FUNCTION_BLOCK Fb_SafetyCheck
VAR_INPUT
END_VAR
VAR_OUTPUT
END_VAR
VAR
	i, j:INT;
	m_checkDelay :ARRAY[1..g_maxNum] OF checkDelay;
	m_checkDelayTime :checkDelayTime;
	m_checkPermit:ARRAY[1..g_maxNum] OF  checkPermit;
	
	m_jntErrFlag:ARRAY[1..g_maxNum,0..g_maxArmJoint,1..3] OF BOOL;
	m_armErrFlag:ARRAY [1..g_maxNum,1..3] OF BOOL;
	m_errCode:UDINT;
	
	
	m_errNumType: ARRAY [1..3] OF INT;
	m_ArrayErrCodeType:ARRAY [1..3] OF ARRAY [0..30] OF UDINT;
	m_ArrayErrCodeTypeTest:ARRAY [1..3] OF ARRAY [0..100] OF UDINT;
	m_armErrCodePopup : ARRAY [1..4] OF ARRAY [0..2] OF UDINT;
	m_armErrCodeRefresh : ARRAY [1..4] OF UINT;
	
	//The fault is sent to the UI at the frequency of 0.1S
	m_errCodeUpdateFlag: ARRAY [1..3] OF BOOL;
	m_errCodeUpdateTon: ARRAY [1..3] OF TON;
	
	m_curJntTorqueIOlast :ARRAY [1..g_maxArmNum] OF vec13di;  
	m_cmdJntPosLast : ARRAY [1..g_maxArmNum] OF vec13d;  
	m_cartCurJntTorqueIOlast :vec8di;  
	m_cartCmdJntPosLast : vec8d;  
	o_ErrCode:ARRAY [1..3] OF UDINT;
		
	m_PromptMassBusy:BOOL;
	m_PromptFlag:ARRAY[1..g_maxNum,1..30] OF UINT;
	m_deleteCode:UDINT;
	
	//joint control error
	m_followErrLimit:vec13d:=[g_largeNum, g_largeNum, 0.010, 4(5*g_deg2Rad), 0.010, 5(170*g_deg2Rad)];
END_VAR


VAR CONSTANT
	m_codeUpdateDelay:TIME:=T#0.1S;
	
	//Fault level: 1 indicates  prompt message, 2 indicates a recoverable fault and 3 indicates an unrecoverable fault
	m_promptMessageLevel : UINT :=1;
	m_rcvLevel : UINT:=2;
	m_unrcvLevel : UINT :=3;
END_VAR

METHOD arrayDeleteFrist : ARRAY [0..30] OF UDINT;
VAR_INPUT
	i_array:ARRAY [0..30] OF UDINT;
END_VAR

VAR
	k:INT;
END_VAR

arrayDeleteFrist[30]:=0;

FOR k:=0 TO 29 BY 1 DO
	arrayDeleteFrist[k]:=i_array[k+1];
END_FOR
END_METHOD

METHOD arrayFILO : ARRAY [0..100] OF  UDINT
VAR_INPUT
	i_array:ARRAY[0..100] OF UDINT;
	i_newData:UDINT;
END_VAR

VAR
	i:INT;
END_VAR

FOR i:=0 TO 20 BY 1 DO
	arrayFILO[i]:=i_array[i];
	IF i_array[i]=0 THEN
		arrayFILO[i]:=i_newData;
		EXIT;
	END_IF
END_FOR
END_METHOD

METHOD cartSafetyCheck : BOOL
VAR_INPUT
	i_armId:UDINT;
	i_safetyCheckVar : checkInputVariable;
	i_cartJointData : ST_CartJointData;
END_VAR


VAR
	k:INT;
END_VAR


//驱动器状态监测、驱动器未连接
FOR i:=1 TO g_maxCartJoint BY 1 DO
	m_checkDelay[i_ArmId].T_cartJntStatusErr[i](IN:= (i_safetyCheckVar.m_cartDriverInput[i].m_statusWord=0 AND m_checkPermit[i_ArmId].m_cartJntStatus[i]), PT:=m_checkDelayTime.Ti_CarJntStatus , Q=> , ET=> );
	IF m_checkDelay[i_ArmId].T_cartJntStatusErr[i].Q THEN
		errCodeAssign(i_ArmId, i_ArmId+3,  0, i, 16#3002 ,m_unrcvLevel );
	END_IF
END_FOR



//关节编码器监测
FOR i:=1 TO g_maxCartJoint BY 1 DO
	m_checkDelay[i_ArmId].T_cartLinkEncErr[i](IN:= (i_safetyCheckVar.m_cartDriverInput[i].m_linkEncoder=g_cartMaxLinkEnc[i] OR i_safetyCheckVar.m_cartDriverInput[i].m_linkEncoder=g_cartMinLinkEnc[i]) AND m_checkPermit[i_ArmId].m_cartJntEncErr[i], PT:=m_checkDelayTime.Ti_CarActSec , Q=> , ET=> );
	IF m_checkDelay[i_ArmId].T_cartLinkEncErr[i].Q THEN
		errCodeAssign(i_ArmId, i_ArmId+3,  0, i, 16#3003 ,m_unrcvLevel );
	END_IF
END_FOR


//驱动器错误检测
FOR i:=1 TO g_maxCartJoint BY 1 DO
	m_checkDelay[i_ArmId].T_cartDriveErr[i](IN:= (i_safetyCheckVar.m_cartDriverInput[i].m_driverError AND 16#20)=32 AND m_checkPermit[i_ArmId].m_cartDriveErr[i] , PT:=m_checkDelayTime.Ti_CarDriveErr , Q=> , ET=> );
	IF m_checkDelay[i_ArmId].T_cartDriveErr[i].Q THEN
		errCodeAssign(i_ArmId, i_ArmId+3,  0, i, 16#3004 ,m_unrcvLevel );
	END_IF
END_FOR



//台车双编码器偏差过大
FOR i:=1 TO g_maxCartJoint BY 1 DO
	m_checkDelay[i_ArmId].T_cartJntEncErr[i](IN:= ABS (i_cartJointData.m_curLinkPos[i]-i_cartJointData.m_curJntPos[i])>g_cartMaxJntEncErr[i] AND m_checkPermit[i_ArmId].m_cartJntEncErr[i], PT:=m_checkDelayTime.Ti_CarDualEncDev , Q=> , ET=> );
	IF m_checkDelay[i_ArmId].T_cartJntEncErr[i].Q THEN
		errCodeAssign(i_ArmId, i_ArmId+3,  0, i, 16#3005 ,m_unrcvLevel );
	END_IF
END_FOR


//关节运动超限位
FOR i:=1 TO g_maxCartJoint BY 1 DO
	m_checkDelay[i_ArmId].T_cartOutOfLimit[i](IN:= (i_cartJointData.m_curJntPos[i]>=g_cartMaxJntPos[i] OR i_cartJointData.m_curJntPos[i]<=g_cartMinJntPos[i]) AND m_checkPermit[i_ArmId].m_cartOutOfLimit[i] , PT:=m_checkDelayTime.Ti_CaroutofLimit , Q=> , ET=> );
	IF m_checkDelay[i_ArmId].T_cartOutOfLimit[i].Q THEN
		errCodeAssign(i_ArmId, i_ArmId+3,  0, i, 16#3006 ,m_unrcvLevel );
	END_IF
END_FOR


//驱动器内部通讯错误
FOR i:=1 TO g_maxCartJoint BY 1 DO
	m_checkDelay[i_ArmId].T_cartCurrentIsNotUpdate[i](IN:= (i_safetyCheckVar.m_cartDriverInput[i].m_current=m_cartCurJntTorqueIOlast[i] AND m_checkPermit[i_ArmId].m_cartCurrentIsNotUpdate[i]), PT:=m_checkDelayTime.Ti_CarTorMotor , Q=> , ET=> );
	IF m_checkDelay[i_ArmId].T_cartCurrentIsNotUpdate[i].Q THEN
		errCodeAssign(i_ArmId, i_ArmId+3,  0, i, 16#3009 ,m_unrcvLevel );
	END_IF
	m_cartCurJntTorqueIOlast[i]:=i_safetyCheckVar.m_cartDriverInput[i].m_current;
END_FOR


//关节跟随误差过大
FOR i:=1 TO g_maxCartJoint BY 1 DO
	m_checkDelay[i_ArmId].T_cartJntFollowErr[i](IN:= ABS(i_cartJointData.m_cmdJntPos[i]- i_cartJointData.m_curJntPos[i])>g_cartMaxJntFollowErr[i]  AND m_checkPermit[i_ArmId].m_cartFollowErr[i], PT:=m_checkDelayTime.Ti_CarFollowDev , Q=> , ET=> );
	IF m_checkDelay[i_ArmId].T_cartJntFollowErr[i].Q THEN
		errCodeAssign(i_ArmId, i_ArmId+3,  0, i, 16#2002 ,m_rcvLevel );
	END_IF
END_FOR


//关节速度监控
FOR i:=1 TO g_maxCartJoint BY 1 DO
	m_checkDelay[i_ArmId].T_cartJntVelErr[i](IN:= ABS(i_cartJointData.m_curJntVel[i])>g_cartMaxJntVel[i] AND m_checkPermit[i_ArmId].m_cartJntVelErr[i], PT:=m_checkDelayTime.Ti_CarJntVel , Q=> , ET=> );
	IF m_checkDelay[i_ArmId].T_cartJntVelErr[i].Q THEN
		errCodeAssign(i_ArmId, i_ArmId+3,  0, i, 16#2003 ,m_rcvLevel );
	END_IF
END_FOR


//电流超限监测
FOR i:=1 TO g_maxCartJoint BY 1 DO
	m_checkDelay[i_ArmId].T_cartJntCurrentErr[i](IN:= ABS(i_cartJointData.m_curJntTrq[i])>g_cartMaxJntCurrent[i] AND m_checkPermit[i_ArmId].m_cartJntCurrentErr[i], PT:=m_checkDelayTime.Ti_CarJntCurrent , Q=> , ET=> );
	IF m_checkDelay[i_ArmId].T_cartJntCurrentErr[i].Q THEN
		errCodeAssign(i_ArmId, i_ArmId+3,  0, i, 16#2005 ,m_rcvLevel );
	END_IF
END_FOR


//Ethercat通讯检测
FOR i:=1 TO g_maxCartJoint BY 1 DO
	IF NOT i_safetyCheckVar.m_cartEtherCATState[i].EtherCATState THEN
		errCodeAssign(i_ArmId, i_ArmId+3,  0, i, 16#2006 ,m_rcvLevel );
	END_IF
END_FOR


//鸣志驱动器错误检测
FOR i:=1 TO g_maxCartJoint BY 1 DO
	m_checkDelay[i_ArmId].T_CarMingzhiDriveErr[i](IN:= (i_safetyCheckVar.m_cartDriverInput[i].m_statusWord AND 16#0F)=15  AND m_checkPermit[i_ArmId].m_cartMZDriveErr[i] , PT:=m_checkDelayTime.Ti_CarMZDriveErr , Q=> , ET=> );
	IF m_checkDelay[i_ArmId].T_CarMingzhiDriveErr[i].Q THEN
		errCodeAssign(i_ArmId, i_ArmId+3,  0, i, 16#2009 ,m_rcvLevel );
	END_IF
END_FOR
END_METHOD

PROPERTY checkPermit : REFERENCE TO ARRAY[1..g_maxNum] OF  checkPermit
GET
checkPermit ref= m_checkPermit;
END_GET
SET
END_SET
END_PROPERTY

METHOD electriAngleDev : DINT
VAR_INPUT
	i_motorElectriAngleDev : DINT;
END_VAR

IF i_motorElectriAngleDev > 50000 THEN
	electriAngleDev := i_motorElectriAngleDev - 65535;
ELSIF i_motorElectriAngleDev < -50000 THEN
	electriAngleDev := i_motorElectriAngleDev + 65535;
ELSE
	electriAngleDev := i_motorElectriAngleDev;
END_IF
END_METHOD

METHOD errCodeAssign : BOOL
VAR_INPUT
	i_armId:UDINT;
	i_errLocation:UDINT;
	i_errCodeMode:UDINT;
	i_errJoint:UDINT;
	i_errID:UDINT;
	i_errFlagID :UINT;
END_VAR
IF m_jntErrFlag[i_armId,i_errJoint,i_errFlagID]=FALSE THEN
	m_jntErrFlag[i_armId,i_errJoint,i_errFlagID]:=TRUE;
	m_errCode:=SHL(i_errLocation,24)+SHL(i_errCodeMode,20)+SHL(i_errJoint,16)+i_errID;
	
	
	IF i_errID>=16#3000 THEN
		m_errNumType[m_unrcvLevel]:=LIMIT(0,m_errNumType[m_unrcvLevel]+1,100);
		m_arrayErrCodeType[m_unrcvLevel][m_errNumType[m_unrcvLevel]]:=m_errCode;
		g_arrayErrCodeArm[i_armId]:=arrayFILO(i_Array:= g_arrayErrCodeArm[i_ArmId], i_NewData:=m_errCode );
		m_armErrFlag[i_armId,m_unrcvLevel]:=TRUE;
		
	ELSIF i_errID>=16#2000 THEN
		m_errNumType[m_rcvLevel]:=LIMIT(0,m_errNumType[m_rcvLevel]+1,100);
		m_arrayErrCodeType[m_rcvLevel][m_errNumType[m_rcvLevel]]:=m_errCode;
		g_arrayErrCodeArm[i_armId]:=arrayFILO(i_Array:= g_arrayErrCodeArm[i_ArmId], i_NewData:=m_errCode );
		m_armErrFlag[i_armId,m_rcvLevel]:=TRUE;
		
	END_IF
END_IF
END_METHOD

METHOD errCodeUpdating :ARRAY [1..3] OF UDINT;
VAR_INPUT
END_VAR

m_errCodeUpdateTon[m_unrcvLevel](IN:= NOT m_errCodeUpdateFlag[3], PT:=m_codeUpdateDelay , Q=> m_errCodeUpdateFlag[3], ET=> );
IF m_errCodeUpdateFlag[m_unrcvLevel] THEN
	IF m_errNumType[m_unrcvLevel]>=1 THEN
		m_ArrayErrCodeType[m_unrcvLevel]:=ArrayDeleteFrist(i_Array:=m_ArrayErrCodeType[3]) ;
		o_ErrCode[m_unrcvLevel]:=m_ArrayErrCodeType[m_unrcvLevel][0] ;
		m_ArrayErrCodeTypeTest[m_unrcvLevel]:=arrayFILO(i_Array:= m_ArrayErrCodeTypeTest[m_unrcvLevel], i_NewData:=o_ErrCode[m_unrcvLevel] );
		m_errNumType[m_unrcvLevel]:=m_errNumType[m_unrcvLevel]-1;
	END_IF
END_IF


m_errCodeUpdateTon[m_rcvLevel](IN:= NOT m_errCodeUpdateFlag[m_rcvLevel], PT:=m_codeUpdateDelay , Q=> m_errCodeUpdateFlag[2], ET=> );
IF m_errCodeUpdateFlag[m_rcvLevel] THEN
	IF m_errNumType[m_rcvLevel]>=1 THEN
		m_ArrayErrCodeType[m_rcvLevel]:=ArrayDeleteFrist(i_Array:=m_ArrayErrCodeType[2]) ;
		o_ErrCode[m_rcvLevel]:=m_ArrayErrCodeType[m_rcvLevel][0] ;
		m_ArrayErrCodeTypeTest[m_rcvLevel]:=arrayFILO(i_Array:= m_ArrayErrCodeTypeTest[m_rcvLevel], i_NewData:=o_ErrCode[m_rcvLevel] );
		m_errNumType[m_rcvLevel]:=m_errNumType[m_rcvLevel]-1;
	END_IF
END_IF
END_METHOD

METHOD errFlagReset : BOOL
VAR_INPUT
END_VAR

FOR i := 1 TO g_maxNum DO
	FOR j :=0 TO g_maxArmJoint DO
		m_jntErrFlag[i, j, 2]:=FALSE;
	END_FOR
	m_armErrFlag[i, 2]:=FALSE;
END_FOR

o_ErrCode[2]:=0;
END_METHOD

METHOD poseErrCheck : vec6d
VAR_INPUT
	i_cmdPose : ST_Frame;
	i_curPose :ST_Frame;
END_VAR

VAR
	posErr,oriErr:Vec3d;
	matT,rotErr:Mat3d;
	errAngle :LREAL;
	errAxis :Vec3d;
	i : INT;
END_VAR
vecSub(i_cmdPose.m_pos, i_curPose.m_pos,posErr);

matTranspose(i_cmdPose.m_rot, matT);
matMultiply(matT,i_curPose.m_rot, rotErr);
rot2AngAxis(rotErr, angle=>errAngle, axis=>errAxis);
vecMultiNum(errAxis, errAngle,oriErr);

FOR i := 1 TO 6 DO
	IF i <= 3 THEN
		poseErrCheck[i] := posErr[i];
	ELSE
		poseErrCheck[i] := oriErr[i];
	END_IF
END_FOR
END_METHOD

METHOD promptMassCode : BOOL
VAR_INPUT
	i_PromptStatus:BOOL;
	i_ArmId:UDINT;
	i_ErrID:UDINT;
	i_ErrLocation:UDINT;
END_VAR
VAR
	m_errStatus : UDINT := 0;
	//error ID , 0-15 bit
	m_errId : UDINT;
	m_arrayErrCode : ARRAY [0..30] OF UDINT;
	m_armErrCode : ARRAY [0..2] OF UDINT;
END_VAR

m_PromptMassBusy:=TRUE;

//prompt flag set true
IF i_PromptStatus=TRUE AND m_PromptFlag[i_ArmId,i_ErrID]=0 THEN
	m_PromptFlag[i_ArmId,i_ErrID]:=1;
END_IF

//
IF i_ErrLocation <= 7 AND i_ErrLocation >= 4 THEN
	m_errStatus := 16#00FF;
ELSE
	m_errStatus := 0;
END_IF
m_errId := i_errID+16#1020;

//output prompt error code
IF m_PromptFlag[i_ArmId,i_ErrID]=1 THEN
	m_ErrCode:=SHL(i_ErrLocation,24)+SHL(m_errStatus,16)+i_errID+16#1020;
	vecFIFO(m_ArrayErrCodeType[1] , m_ErrCode , m_arrayErrCode );
	m_ArrayErrCodeType[1]:=m_arrayErrCode;
	IF (m_ErrCode AND 16#00FF0000) = 16#00FF0000 THEN
		vecFIFO(m_armErrCodePopup[i_armId] , m_ErrCode , m_armErrCode );
		m_armErrCodePopup[i_armId] := m_armErrCode;
		m_armErrCodeRefresh[i_armId] := 1;
	END_IF
	m_PromptFlag[i_ArmId,i_ErrID]:=2;
END_IF

//clear prompt error code
IF m_PromptFlag[i_ArmId,i_ErrID]=2 AND i_PromptStatus=FALSE THEN
	m_deleteCode:=SHL(i_ErrLocation,24)+SHL(m_errStatus,16)+i_ErrID+16#1020;
	vecDeleteInput(m_ArrayErrCodeType[1] , m_deleteCode , m_arrayErrCode);
	m_ArrayErrCodeType[1] := m_arrayErrCode;
	IF (m_deleteCode AND 16#00FF0000)  = 16#00FF0000 THEN
		vecDeleteInput(m_armErrCodePopup[i_armId] , m_deleteCode , m_armErrCode );
		m_armErrCodePopup[i_armId] := m_armErrCode;
		m_armErrCodeRefresh[i_armId] := 2;
	END_IF
	//ArrayDeleteInput(i_Array:= m_ArrayErrCodeType[1], i_DeleteCode:=m_deleteCode , o_Array=> m_ArrayErrCodeType[1]);
	m_PromptFlag[i_ArmId,i_ErrID]:=0;
END_IF
o_ErrCode[1]:=m_ArrayErrCodeType[1][0];
m_PromptMassBusy:=FALSE;
END_METHOD

METHOD rcpErrCheck : BOOL
VAR_INPUT
	i_cmdPos : Vec3d;
	i_curPos : Vec3d;
END_VAR
VAR_IN_OUT
	r_errCount:INT;
	r_posErr :Vec3d;
END_VAR

VAR
	err:Vec3d;
END_VAR
vecSub(i_cmdPos, i_curPos,err);
r_posErr:=err;

IF  (norm(err)>g_rcpDeviationThres) THEN
	r_errCount:= r_errCount +1;
ELSE 
	r_errCount:=0;
END_IF
rcpErrCheck := r_errCount >= g_faultTriggerCounts;
END_METHOD

METHOD setupSafetyCheck : BOOL
VAR_INPUT
	i_armId:UDINT;
	i_safetyCheckVar :ARRAY[1..g_maxNum] OF checkInputVariable;
	i_setupJointData : ST_SetupJointData;
END_VAR

VAR
	k:INT;
END_VAR


//驱动器状态监测、驱动器未连接
FOR i:=1 TO g_setupJntNum BY 1 DO
	m_checkDelay[i_ArmId].T_jntStatusErr[i](IN:= (i_safetyCheckVar[i_ArmId].m_setupDriverInput[i].m_statusWord=0 AND m_checkPermit[i_ArmId].m_jntStatusErr[i]), PT:=m_checkDelayTime.Ti_jntStatusErr , Q=> , ET=> );
	IF m_checkDelay[i_ArmId].T_jntStatusErr[i].Q THEN
		errCodeAssign(i_ArmId, i_ArmId+3,  0, i, 16#3002 ,m_unrcvLevel );
	END_IF
END_FOR



//关节编码器监测
FOR i:=1 TO g_setupJntNum BY 1 DO
	m_checkDelay[i_ArmId].T_linkEncErr[i](IN:= (i_safetyCheckVar[i_ArmId].m_setupDriverInput[i].m_linkEncoder=g_maxLinkEnc[i] OR i_safetyCheckVar[i_ArmId].m_setupDriverInput[i].m_linkEncoder=g_minLinkEnc[i]) AND m_checkPermit[i_ArmId].m_linkEncErr[i], PT:=m_checkDelayTime.Ti_linkEncErr , Q=> , ET=> );
	IF m_checkDelay[i_ArmId].T_linkEncErr[i].Q THEN
		errCodeAssign(i_ArmId, i_ArmId+3,  0, i,  16#3003 ,m_unrcvLevel );
	END_IF
END_FOR


//驱动器错误检测
FOR i:=1 TO g_setupJntNum BY 1 DO
	m_checkDelay[i_ArmId].T_DriveErr[i](IN:= (i_safetyCheckVar[i_ArmId].m_setupDriverInput[i].m_driverError AND 16#20)=g_driveErrWord AND m_checkPermit[i_ArmId].m_driveErr[i] , PT:=m_checkDelayTime.Ti_driveErr , Q=> , ET=> );
	IF m_checkDelay[i_ArmId].T_DriveErr[i].Q THEN
		errCodeAssign(i_ArmId, i_ArmId+3,  0, i, 16#3004 ,m_unrcvLevel );
	END_IF
END_FOR


//双编码器偏差过大检测
FOR i:=1 TO g_setupJntNum BY 1 DO
	m_checkDelay[i_ArmId].T_armJntEncErr[i](IN:= ABS(i_setupJointData.m_curLinkPos[i_armId][i]-i_setupJointData.m_curJntPos[i_armId][i])>=g_armMaxJntEncErr[i] AND m_checkPermit[i_ArmId].m_armJntEncErr[i], PT:=m_checkDelayTime.Ti_armJntEncErr , Q=> , ET=> );
	IF m_checkDelay[i_ArmId].T_armJntEncErr[i].Q THEN
		errCodeAssign( i_ArmId, i_ArmId+3,  0, i, 16#3005, m_unrcvLevel );
	END_IF
END_FOR


//关节运动超限位
FOR i:=1 TO g_setupJntNum BY 1 DO
	m_checkDelay[i_ArmId].T_outOfLimit[i](IN:= (i_setupJointData.m_curJntPos[i_armId][i]>=(g_maxJntPos[i_armId,i]+g_armJntPosLimitBuffer[i]) OR i_setupJointData.m_curJntPos[i_armId][i]<=(g_minJntPos[i_armId,i]-g_armJntPosLimitBuffer[i])) AND m_checkPermit[i_ArmId].m_outOfLimit[i] , PT:=m_checkDelayTime.Ti_outofLimit , Q=> , ET=> );
	IF m_checkDelay[i_ArmId].T_outOfLimit[i].Q THEN
		errCodeAssign(i_ArmId, i_ArmId+3,  0, i, 16#3006, m_unrcvLevel );
	END_IF
END_FOR


//电机电角度偏差
FOR i:=1 TO g_setupJntNum BY 1 DO
	IF ABS(electriAngleDev(i_safetyCheckVar[i_armId].m_setupDriverInput[i].m_electriAngleDev))> g_motPhieErrLimit  AND m_checkPermit[i_ArmId].m_motPhieErr[i] THEN
		errCodeAssign(i_ArmId, i_ArmId+3,  0, i, 16#3008, m_unrcvLevel );
	END_IF
END_FOR


//驱动器内部通讯错误
FOR i:=1 TO g_setupJntNum BY 1 DO
	m_checkDelay[i_ArmId].T_currentIsNotUpdate[i](IN:= (i_safetyCheckVar[i_ArmId].m_setupDriverInput[i].m_current=m_curJntTorqueIOlast[i_ArmId][i] AND m_checkPermit[i_ArmId].m_currentIsNotUpdate[i]), PT:=m_checkDelayTime.Ti_currentIsNotUpdate , Q=> , ET=> );
	IF  m_checkDelay[i_ArmId].T_currentIsNotUpdate[i].Q THEN
		errCodeAssign(i_ArmId, i_ArmId+3,  0, i, 16#3009 ,m_unrcvLevel );
	END_IF
	m_curJntTorqueIOlast[i_ArmId][i]:=i_safetyCheckVar[i_ArmId].m_setupDriverInput[i].m_current;
END_FOR


//关节跟随误差过大
FOR i:=1 TO g_setupJntNum BY 1 DO
	m_checkDelay[i_ArmId].T_armJntFollowErr[i](IN:= ABS(i_setupJointData.m_cmdJntPos[i_armId][i]- i_setupJointData.m_curJntPos[i_armId][i])>g_armMaxJntFollowErr[i]  AND m_checkPermit[i_ArmId].m_armJntFollowErr[i], PT:=m_checkDelayTime.Ti_armJntFollowErr , Q=> , ET=> );
	IF m_checkDelay[i_ArmId].T_armJntFollowErr[i].Q THEN
		errCodeAssign(i_ArmId, i_ArmId+3,  0, i, 16#2002, m_rcvLevel );
	END_IF
END_FOR


//关节速度监控
FOR i:=1 TO g_setupJntNum BY 1 DO
	m_checkDelay[i_ArmId].T_jntVelErr[i](IN:= ABS (i_setupJointData.m_curJntVel[i_armId][i])>g_safetyJntVel[i] AND m_checkPermit[i_ArmId].m_jntVelErr[i], PT:=m_checkDelayTime.Ti_jntVelErr , Q=> , ET=> );
	IF m_checkDelay[i_ArmId].T_jntVelErr[i].Q THEN
		errCodeAssign(i_ArmId, i_ArmId+3,  0, i, 16#2003, m_rcvLevel );
	END_IF
END_FOR



//电流超限监测
FOR i:=1 TO g_setupJntNum BY 1 DO
	m_checkDelay[i_ArmId].T_jntCurrentErr[i](IN:= ABS(i_setupJointData.m_rawJntCurrent[i_armId][i])>g_maxJntCurrent[i] AND m_checkPermit[i_ArmId].m_jntCurrentErr[i], PT:=m_checkDelayTime.Ti_jntCurrentErr , Q=> , ET=> );
	IF m_checkDelay[i_ArmId].T_jntCurrentErr[i].Q THEN
		errCodeAssign(i_ArmId, i_ArmId+3,  0, i, 16#2005, m_rcvLevel );
	END_IF
END_FOR


//Ethercat通讯检测
FOR i:=1 TO g_setupJntNum BY 1 DO
	IF NOT i_safetyCheckVar[i_ArmId].m_EtherCATState[i].EtherCATState THEN
		errCodeAssign(i_ArmId, i_ArmId+3, 0, i, 16#2006, m_rcvLevel );
	END_IF
END_FOR


//不动点发生变化监控
m_checkDelay[i_ArmId].T_FixedPointErr(IN:=  i_safetyCheckVar[i_ArmId].m_rcpCheck AND m_checkPermit[i_ArmId].m_fixedPointErr, PT:=m_checkDelayTime.Ti_FixedPointErr , Q=> , ET=> );
IF m_checkDelay[i_ArmId].T_FixedPointErr.Q THEN
	errCodeAssign(i_ArmId, i_ArmId+3,  0, 0, 16#2007, m_rcvLevel );
END_IF


//目标位置指令突变检测
FOR i:=1 TO g_setupJntNum BY 1 DO
	IF (i_setupJointData.m_cmdJntPos[i_armId][i]-m_cmdJntPosLast[i_ArmId][i])>g_maxJntCmdSalta[i] AND m_checkPermit[i_ArmId].m_cmdJntSaltation[i] THEN
		errCodeAssign(i_armId, i_ArmId+3, 0, i, 16#2008, m_rcvLevel );
	END_IF
	m_cmdJntPosLast[i_armId][i] := i_setupJointData.m_cmdJntPos[i_armId][i];
END_FOR


//Deviation between command current and feedback current
FOR i:=1 TO g_setupJntNum BY 1 DO
	IF ABS(i_safetyCheckVar[i_armId].m_slaveDriverOutput[i].m_cmdCurrent-i_safetyCheckVar[i_armId].m_slaveDriverInput[i].m_current)> g_jntCurrentCtrlLimit[i]  AND m_checkPermit[i_armId].m_jntCurrentCtrlErr[i] THEN
		errCodeAssign(i_armId, i_armId+3, 0, i, 16#200B, m_rcvLevel );
	END_IF
END_FOR


//motor encoder mutation detection
FOR i:=1 TO g_setupJntNum BY 1 DO
	IF (i_safetyCheckVar[i_armId].m_motorEncoderSaltaValue[i])>g_maxJntCurSalta[i] THEN
		errCodeAssign(i_armId, i_ArmId+3, 0, i, 16#200C, m_rcvLevel );
	END_IF
END_FOR
END_METHOD

METHOD slaveSafetyCheck : BOOL
VAR_INPUT
	i_armId:UDINT;
	i_safetyCheckVar :ARRAY[1..g_maxNum] OF checkInputVariable;
	i_slaveJointData : ST_SlaveJointData;
END_VAR
//驱动器状态监测、驱动器未连接
FOR i:=1 TO g_sJntNum BY 1 DO
	m_checkDelay[i_ArmId].T_jntStatusErr[i+g_setupJntNum](IN:= (i_safetyCheckVar[i_ArmId].m_slaveDriverInput[i].m_statusWord=0 AND m_checkPermit[i_ArmId].m_jntStatusErr[i+g_setupJntNum]), PT:=m_checkDelayTime.Ti_jntStatusErr , Q=> , ET=> );
	IF m_checkDelay[i_ArmId].T_jntStatusErr[i+g_setupJntNum].Q  THEN
		errCodeAssign(i_ArmId, i_ArmId+3,  0, i+g_setupJntNum, 16#3002 ,m_unrcvLevel );
	END_IF
END_FOR



//关节编码器监测
FOR i:=1 TO g_sJntNum BY 1 DO
	m_checkDelay[i_ArmId].T_linkEncErr[i+g_setupJntNum](IN:= (i_safetyCheckVar[i_ArmId].m_slaveDriverInput[i].m_linkEncoder=g_maxLinkEnc[i] OR i_safetyCheckVar[i_ArmId].m_slaveDriverInput[i].m_linkEncoder=g_minLinkEnc[i]) AND m_checkPermit[i_ArmId].m_linkEncErr[i], PT:=m_checkDelayTime.Ti_linkEncErr , Q=> , ET=> );
	IF m_checkDelay[i_ArmId].T_linkEncErr[i+g_setupJntNum].Q THEN
		errCodeAssign(i_ArmId, i_ArmId+3,  0, i+g_setupJntNum,  16#3003 ,m_unrcvLevel );
	END_IF
END_FOR


//驱动器错误检测
FOR i:=1 TO g_sJntNum BY 1 DO
	m_checkDelay[i_ArmId].T_DriveErr[i+g_setupJntNum](IN:= (i_safetyCheckVar[i_ArmId].m_slaveDriverInput[i].m_driverError AND 16#20)=g_driveErrWord AND m_checkPermit[i_ArmId].m_driveErr[i] , PT:=m_checkDelayTime.Ti_driveErr , Q=> , ET=> );
	IF m_checkDelay[i_ArmId].T_DriveErr[i+g_setupJntNum].Q THEN
		errCodeAssign(i_ArmId, i_ArmId+3,  0, i+g_setupJntNum, 16#3004 ,m_unrcvLevel );
	END_IF
END_FOR


//双编码器偏差过大检测
FOR i:=1 TO g_sJntNum-5 BY 1 DO
	m_checkDelay[i_ArmId].T_armJntEncErr[i+g_setupJntNum](IN:= ABS(i_slaveJointData.m_curLinkPos[i_armId][i]-i_slaveJointData.m_curJntPos[i_armId][i])>=g_armMaxJntEncErr[i+g_setupJntNum] AND m_checkPermit[i_ArmId].m_armJntEncErr[i+g_setupJntNum], PT:=m_checkDelayTime.Ti_armJntEncErr , Q=> , ET=> );
	IF m_checkDelay[i_ArmId].T_armJntEncErr[i+g_setupJntNum].Q THEN
		errCodeAssign( i_ArmId, i_ArmId+3,  0, i+g_setupJntNum, 16#3005, m_unrcvLevel );
	END_IF
END_FOR


//关节运动超限位
FOR i:=1 TO g_sJntNum BY 1 DO
	m_checkDelay[i_ArmId].T_outOfLimit[i+g_setupJntNum](IN:= (i_slaveJointData.m_curJntPos[i_armId][i]>=(g_maxJntPos[i_armId,i+g_setupJntNum]+g_armJntPosLimitBuffer[i+g_setupJntNum]) OR i_slaveJointData.m_curJntPos[i_armId][i]<=(g_minJntPos[i_armId,i+g_setupJntNum]-g_armJntPosLimitBuffer[i+g_setupJntNum])) AND m_checkPermit[i_ArmId].m_outOfLimit[i+g_setupJntNum] , PT:=m_checkDelayTime.Ti_outofLimit , Q=> , ET=> );
	IF m_checkDelay[i_ArmId].T_outOfLimit[i+g_setupJntNum].Q THEN
		errCodeAssign(i_ArmId, i_ArmId+3,  0, i+g_setupJntNum, 16#3006, m_unrcvLevel );
	END_IF
END_FOR


//电机电角度偏差
FOR i:=1 TO g_sJntNum BY 1 DO
	IF ABS(electriAngleDev(i_safetyCheckVar[i_armId].m_slaveDriverInput[i].m_electriAngleDev))> g_motPhieErrLimit  AND m_checkPermit[i_ArmId].m_motPhieErr[i+g_setupJntNum] THEN
		errCodeAssign(i_ArmId, i_ArmId+3,  0, i+g_setupJntNum, 16#3008, m_unrcvLevel );
	END_IF
END_FOR


//驱动器内部通讯错误
FOR i:=1 TO g_sJntNum BY 1 DO
	m_checkDelay[i_ArmId].T_currentIsNotUpdate[i+g_setupJntNum](IN:= (i_safetyCheckVar[i_ArmId].m_slaveDriverInput[i].m_current=m_curJntTorqueIOlast[i_ArmId][i+g_setupJntNum] AND m_checkPermit[i_ArmId].m_currentIsNotUpdate[i+g_setupJntNum]), PT:=m_checkDelayTime.Ti_currentIsNotUpdate , Q=> , ET=> );
	IF  m_checkDelay[i_ArmId].T_currentIsNotUpdate[i+g_setupJntNum].Q THEN
		errCodeAssign(i_ArmId, i_ArmId+3,  0, i+g_setupJntNum, 16#3009 ,m_unrcvLevel );
	END_IF
	m_curJntTorqueIOlast[i_ArmId][i+g_setupJntNum]:=i_safetyCheckVar[i_ArmId].m_slaveDriverInput[i].m_current;
END_FOR


//关节跟随误差过大---1028
FOR i:=1 TO g_sJntNum BY 1 DO
	(*
	m_checkDelay[i_ArmId].T_armJntFollowErr[i+g_setupJntNum](IN:= ABS(i_slaveJointData.m_cmdJntPos[i_armId][i]- i_slaveJointData.m_curJntPos[i_armId][i])>g_armMaxJntFollowErr[i+g_setupJntNum]  AND m_checkPermit[i_ArmId].m_armJntFollowErr[i+g_setupJntNum], PT:=m_checkDelayTime.Ti_armJntFollowErr , Q=> , ET=> );
	IF m_checkDelay[i_ArmId].T_armJntFollowErr[i+g_setupJntNum].Q THEN
		errCodeAssign(i_ArmId, i_ArmId+3,  0, i+g_setupJntNum, 16#2002, m_rcvLevel );
	END_IF
	*)
	
	//update the control error limit
	IF (SlaveArmControl.m_slaveRobot.m_stiffChanged[i_ArmId]=TRUE) THEN
		m_followErrLimit:=g_armMaxJntFollowErrSoftStiff;
	ELSE
		m_followErrLimit:=g_armMaxJntFollowErr;
	END_IF
	
	//check
	m_checkDelay[i_ArmId].T_armJntFollowErr[i+g_setupJntNum](IN:= ABS(i_slaveJointData.m_cmdJntPos[i_armId][i]- i_slaveJointData.m_curJntPos[i_armId][i])>m_followErrLimit[i+g_setupJntNum]  AND m_checkPermit[i_ArmId].m_armJntFollowErr[i+g_setupJntNum], PT:=m_checkDelayTime.Ti_armJntFollowErr , Q=> , ET=> );
	IF m_checkDelay[i_ArmId].T_armJntFollowErr[i+g_setupJntNum].Q THEN
		errCodeAssign(i_ArmId, i_ArmId+3,  0, i+g_setupJntNum, 16#2002, m_rcvLevel );
	END_IF	
END_FOR


//关节速度监控
FOR i:=1 TO g_sJntNum-5 BY 1 DO
	m_checkDelay[i_ArmId].T_jntVelErr[i+g_setupJntNum](IN:= ABS (i_slaveJointData.m_curJntVel[i_armId][i])>g_safetyJntVel[i+g_setupJntNum] AND m_checkPermit[i_ArmId].m_jntVelErr[i+g_setupJntNum], PT:=m_checkDelayTime.Ti_jntVelErr , Q=> , ET=> );
	IF m_checkDelay[i_ArmId].T_jntVelErr[i+g_setupJntNum].Q THEN
		errCodeAssign(i_ArmId, i_ArmId+3,  0, i+g_setupJntNum, 16#2003, m_rcvLevel );
	END_IF
END_FOR


// TODO: replaced with cartesin twist check
//笛卡尔空间指令与位置偏差检测
//FOR i:=1 TO 6 BY 1 DO
//	m_checkDelay[i_ArmId].T_spacePoseErr[i](IN:= i_safetyCheckVar[i_ArmId].m_spacePoseErr[i]> g_maxCartPoseErr[i] AND m_checkPermit[i_ArmId].m_spacePoseErr[i], PT:=m_checkDelayTime.Ti_spacePoseErr , Q=> , ET=> );
//	IF m_checkDelay[i_ArmId].T_spacePoseErr[i].Q THEN
//		errCodeAssign(i_ArmId, i_ArmId+3, 1, i, 16#2004, m_rcvLevel );
//	END_IF
//END_FOR


//电流超限监测
FOR i:=1 TO g_sJntNum BY 1 DO
	m_checkDelay[i_ArmId].T_jntCurrentErr[i+g_setupJntNum](IN:= ABS(i_slaveJointData.m_rawJntCurrent[i_armId][i])>g_maxJntCurrent[i+g_setupJntNum] AND m_checkPermit[i_ArmId].m_jntCurrentErr[i+g_setupJntNum], PT:=m_checkDelayTime.Ti_jntCurrentErr , Q=> , ET=> );
	IF m_checkDelay[i_ArmId].T_jntCurrentErr[i+g_setupJntNum].Q THEN
		errCodeAssign(i_ArmId, i_ArmId+3,  0, i+g_setupJntNum, 16#2005, m_rcvLevel );
	END_IF
END_FOR


//Ethercat通讯检测
FOR i:=1 TO g_sJntNum BY 1 DO
	IF NOT i_safetyCheckVar[i_ArmId].m_EtherCATState[i+g_setupJntNum].EtherCATState THEN
		errCodeAssign(i_ArmId, i_ArmId+3, 0, i+g_setupJntNum, 16#2006, m_rcvLevel );
	END_IF
END_FOR


//目标位置指令突变检测
FOR i:=1 TO g_sJntNum BY 1 DO
	m_checkDelay[i_ArmId].T_jntCmdSalta[i+g_setupJntNum](IN:= m_checkPermit[i_ArmId].m_cmdJntSaltation[i+g_setupJntNum], PT:=m_checkDelayTime.Ti_jntCmdSaltationErr , Q=> , ET=> );
	IF m_checkDelay[i_ArmId].T_jntCmdSalta[i+g_setupJntNum].Q THEN
		IF (i_slaveJointData.m_cmdJntPos[i_armId][i]-m_cmdJntPosLast[i_ArmId][i+g_setupJntNum])>g_maxJntCmdSalta[i+g_setupJntNum] THEN
			errCodeAssign(i_ArmId, i_ArmId+3, 0, i+g_setupJntNum, 16#2008, m_rcvLevel );
		END_IF
	END_IF
	m_cmdJntPosLast[i_ArmId][i+g_setupJntNum] := i_slaveJointData.m_cmdJntPos[i_armId][i];
END_FOR


//Deviation between command current and feedback current
//FOR i:=1 TO g_sJntNum BY 1 DO
//	IF ABS(i_safetyCheckVar[i_armId].m_slaveDriverOutput[i].m_cmdCurrent-i_safetyCheckVar[i_armId].m_slaveDriverInput[i].m_current)> g_jntCurrentCtrlLimit[i+g_setupJntNum]  AND m_checkPermit[i_armId].m_jntCurrentCtrlErr[i+g_setupJntNum] THEN
//		errCodeAssign(i_armId, i_armId+3, 0, i+g_setupJntNum, 16#200B, m_rcvLevel );
//	END_IF
//END_FOR


//motor encoder mutation detection
FOR i:=1 TO g_sJntNum BY 1 DO
	IF (i_safetyCheckVar[i_armId].m_motorEncoderSaltaValue[i+g_setupJntNum])>g_maxJntCurSalta[i+g_setupJntNum] THEN
		errCodeAssign(i_armId, i_ArmId+3, 0, i+g_setupJntNum, 16#200C, m_rcvLevel );
	END_IF
END_FOR


//器械张开角度过大或过小
IF (i_safetyCheckVar[i_ArmId].m_instruOpenAngle> g_maxInstruOpen OR i_safetyCheckVar[i_ArmId].m_instruOpenAngle< 0) AND m_checkPermit[i_ArmId].m_instruOpenAngle THEN
	errCodeAssign(i_ArmId, i_ArmId+3, 0, 0, 16#200D, m_rcvLevel );
END_IF
END_METHOD

METHOD systemSafetyCheck : BOOL
VAR_INPUT
	i_armId:UDINT;
	i_safetyCheckVar :ARRAY[1..g_maxNum] OF checkInputVariable;
	i_cartJointData : ST_CartJointData;
	i_setupJointData : ST_SetupJointData;
	i_slaveJointData : ST_SlaveJointData;
END_VAR

VAR
	k:INT;
END_VAR

IF i_armId =g_cartNum THEN 
	//cart safrty check
	cartSafetyCheck(i_armId,i_safetyCheckVar[i_armId],i_cartJointData);
ELSE
	//EmergencyStopButton
	IF NOT i_safetyCheckVar[i_ArmId].EmergencyStop OR m_jntErrFlag[i_armId,0,3] THEN
		errCodeAssign(i_ArmId, 16#0C, 0, 0, 16#3001, m_unrcvLevel);
		RETURN;
	END_IF
	//setup arms safety check
	setupSafetyCheck(i_armId,i_safetyCheckVar,i_setupJointData);
	//slave arms safety check
	slaveSafetyCheck(i_armId,i_safetyCheckVar,i_slaveJointData);
END_IF

//StopButton
IF NOT i_safetyCheckVar[i_ArmId].SlaveStopButton OR i_safetyCheckVar[i_ArmId].PCStopButton=0 OR i_safetyCheckVar[i_ArmId].MasterStopButton THEN
	errCodeAssign(i_ArmId, 16#0C, 0, 0, 16#2001, m_rcvLevel );
END_IF

//prompt message
FOR i:=1 TO 30 BY 1 DO
	PromptMassCode( i_safetyCheckVar[i_ArmId].m_promptStatus[i], i_ArmId,  i,  i_safetyCheckVar[i_ArmId].m_promptLocation[i]);
END_FOR
END_METHOD

METHOD vecDeleteInput : BOOL
VAR_IN_OUT CONSTANT
	vecA :ARRAY[*] OF UDINT;
END_VAR

VAR_INPUT
	i_deleteCode :UDINT;
END_VAR

VAR_IN_OUT
	vecB : ARRAY[*] OF UDINT;
END_VAR

VAR
	m :DINT;
	i :DINT;
	Falg:BOOL;
END_VAR
m:=UPPER_BOUND(vecA,1);

FOR i:=0 TO m BY 1 DO 
	IF vecA[i]=i_DeleteCode THEN
		Falg:=TRUE;
	END_IF
	
	IF Falg=TRUE THEN
		vecB[i]:=vecA[i+1];
	ELSE
		vecB[i]:=vecA[i];
	END_IF
END_FOR
vecB[m]:=0;
END_METHOD

METHOD vecFIFO : BOOL
VAR_IN_OUT CONSTANT
	vecA :ARRAY[*] OF UDINT;
END_VAR

VAR_INPUT
	i_newData :UDINT;
END_VAR

VAR_IN_OUT
	vecB : ARRAY[*] OF UDINT;
END_VAR

VAR
	m :DINT;
	i :DINT;
END_VAR
m:=UPPER_BOUND(vecA,1);

FOR i:=0 TO m DO
	vecB[i+1]:=vecA[i];
END_FOR

vecB[0]:=i_newData;
END_METHOD

END_FUNCTION_BLOCK

(* stored: Version 1.1.0.1, ProductVersion 3.1.4024.11
   POU Fb_SafetyCheck: Id {d7e5b419-2971-4dae-96a7-39fe3a1a6245}, SpecialFunc None
   Folder interface: Id {17cc820b-439e-4bcd-b035-470b65e01b6b}
   Method arrayDeleteFrist: Id {00e49c9f-cbe8-4b26-b05a-c4b6acb31969}
   Method arrayFILO: Id {26262d95-ef1c-497d-b548-c28fcd1771c9}
   Method cartSafetyCheck: Id {64489d60-54d3-406d-a82e-df5d6a98f0f1}
   Property checkPermit: Id {4ac5d9ef-e4e1-4258-a3b3-a263171adb15}
   Get Get: Id {5a600670-0a2f-4560-9a82-9a30fff97e6d}
   Set Set: Id {06536298-2ca0-4bed-b4ee-b29089d28252}
   Method electriAngleDev: Id {8c2ea40a-ba18-4d9e-8d1f-4ea5c9f320b3}
   Method errCodeAssign: Id {c6bfedc5-fddc-4db6-ba7d-64971d20a433}
   Method errCodeUpdating: Id {0b3c9bb2-9217-4fc9-b998-e4a685172889}
   Method errFlagReset: Id {2f8c115b-de2b-4c35-92d2-fdbed32dcf1f}
   Method poseErrCheck: Id {634b1f68-028c-4865-89df-6d37274cf53c}
   Method promptMassCode: Id {97898266-aa01-4d86-bccd-f23152d91670}
   Method rcpErrCheck: Id {1ac09358-1d04-48f7-ae97-15cd7273ced0}
   Method setupSafetyCheck: Id {09c2f1a9-8e0a-4d09-a292-1a371f055e17}
   Method slaveSafetyCheck: Id {1102e175-6107-4706-a6ad-ea5e8fc76a1b}
   Method systemSafetyCheck: Id {7874ef26-88d5-4eb7-8db9-4fa17a2dd1f0}
   Method vecDeleteInput: Id {e506aae7-9713-4864-8cb2-3b20c292dbc5}
   Method vecFIFO: Id {5b91c1fa-b44e-445d-b440-100929259021} *)
